PROGRAM InterfaceTesting
VAR
	fbParent : FB_Object(FALSE,1);
	fbChild : FB_ObjectExt(FALSE,2);
	fbSecond : FB_SecondObject;
	
	//Declaration interface assignment
	iParent : ITF_Object := fbParent;
	iChild : ITF_ObjectExt;
	
	//Declaration interface injected through constructor
	fbThird : FB_ThirdObject(ParentObject := fbParent);
	bCastResult : BOOL;
END_VAR

//Interface assignment in code
iChild := fbChild;

//Interface in property takes the parent interface
//passing child class here
fbSecond.ParentObject := fbChild;

//use method call to test cast
//child passed in using parent interface, need to cast to use child interface methods
bCastResult := fbSecond.AttemptCast();

END_PROGRAM

(* stored: Version 1.1.0.1, ProductVersion 3.1.4024.11
   POU InterfaceTesting: Id {99f5130b-9b5f-4b2d-99a7-ef2887d70542}, SpecialFunc None *)
